PROGRAM MAIN
VAR
END_VAR

ModbusTCP();

END_PROGRAM

(* stored: Version 1.1.0.1, ProductVersion 3.1.4026.18
   POU MAIN: Id {8a81df4b-51d6-40e4-803a-6781ac8ddcf3}, SpecialFunc None *)
